FUNCTION_BLOCK CfbTop
  (* Standard: 61499-2 *)
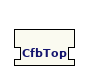
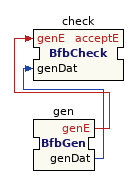
  FBS
    check : BfbCheck;
    gen : BfbGen;
  END_FBS
  EVENT_CONNECTIONS
    gen.genE TO check.genE;
  END_CONNECTIONS
  DATA_CONNECTIONS
    gen.genDat TO check.genDat;
  END_CONNECTIONS
END_FUNCTION_BLOCK
